(* CODESYS project Projeto_Prensa.project

Project tree, tasks and I/O mapping:
  Device : CODESYS Control Win V3, 3S - Smart Software Solutions GmbH, order no. 305021, version 3.5.11.30
    application Application
      libraries: Standard, * (System)
      task MainTask (cyclic, interval t#20ms, priority 1) calls PLC_PRG
      task VISU_TASK (cyclic, interval 100 ms, priority 31) calls VisuElems.Visu_Prg
      program PLC_PRG [LD]
      Symbols
      visualisation Visualization
  libraries: VisuSymbols, 3.5.10.0 (System)
  text list GlobalTextList
*)

// Device/Application/PLC_PRG
PROGRAM PLC_PRG
VAR
	SENSOR1: REAL; //SENSOR DE PRESSÃO M1
	SENSOR2: REAL; //SENSOR DE PRESSÃO M2
	SENSOR3: REAL; //SENSOR DE PRESSÃO P1
	PRES1: REAL; //PRESSÃO M1
	PRES2: REAL; //PRESSÃO M2
	PRES3: REAL; //PRESSÃO P1
	AL1: BOOL; // ALARME PRES1
	AL2: BOOL; // ALARME PRES2
	AL3: BOOL; // ALARME PRES3
	I7: BOOL; //B1
	I0: BOOL; //S1
	I1: BOOL; //S2
	I2: BOOL; //S3
	I3: BOOL; //S4
	I4: BOOL; //S5
	I5: BOOL; //S6
	M0: BOOL; //K1
	M1: BOOL; //K2
	M2: BOOL; //K3
	M3: BOOL; //K4
	M4: BOOL; //K5
	Q0: BOOL; //Y1
	Q1: BOOL; //Y2
	Q2: BOOL; //Y3
	Q3: BOOL; //Y4
	Q4: BOOL; //Y5
	ED0: BYTE;  // Byte para fluidsim - ENTRADAS
	AB0: BYTE;  // Byte para fluidsim - SAIDAS
END_VAR
VAR // added by the converter: edge detectors and wires of the graphical bodies
    _w1 : BOOL;
END_VAR

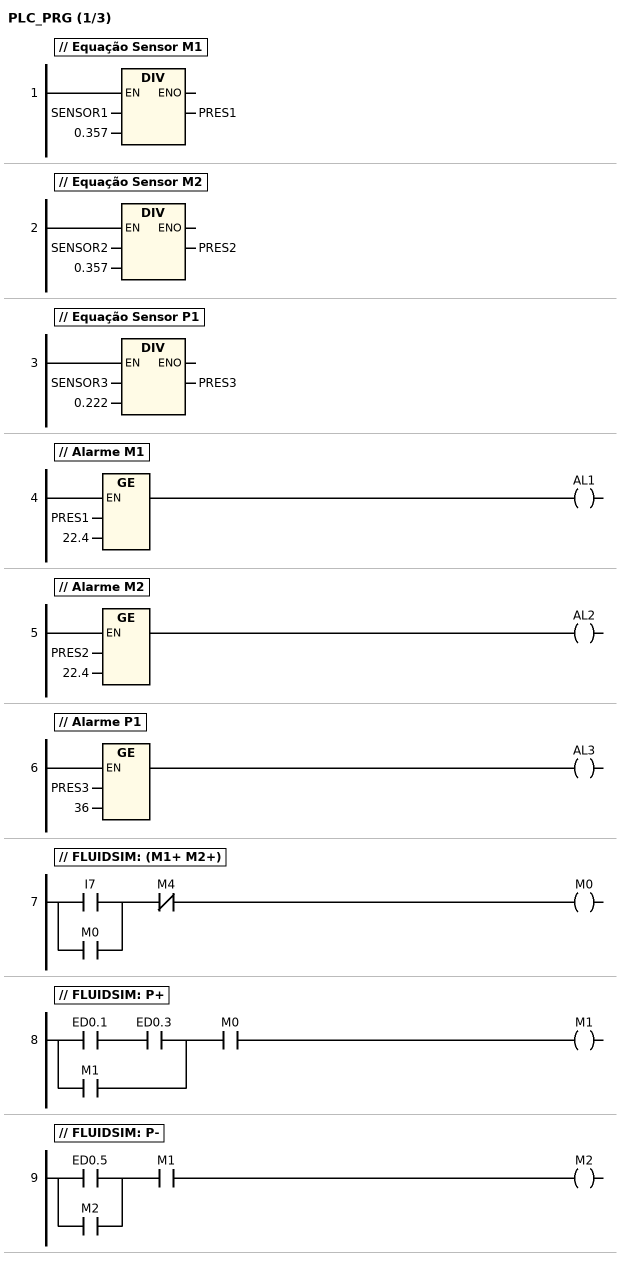
// NETWORK 1
// label: // Equação Sensor M1
PRES1 := SENSOR1 / 0.357;

// NETWORK 2
// label: // Equação Sensor M2
PRES2 := SENSOR2 / 0.357;

// NETWORK 3
// label: // Equação Sensor P1
PRES3 := SENSOR3 / 0.222;

// NETWORK 4
// label: // Alarme M1
AL1 := PRES1 >= 22.4;

// NETWORK 5
// label: // Alarme M2
AL2 := PRES2 >= 22.4;

// NETWORK 6
// label: // Alarme P1
AL3 := PRES3 >= 36;

// NETWORK 7
// label: // FLUIDSIM: (M1+ M2+)
M0 := (I7 OR M0) AND NOT M4;

// NETWORK 8
// label: // FLUIDSIM: P+
M1 := (ED0.1 AND ED0.3 OR M1) AND M0;

// NETWORK 9
// label: // FLUIDSIM: P-
M2 := (ED0.5 OR M2) AND M1;

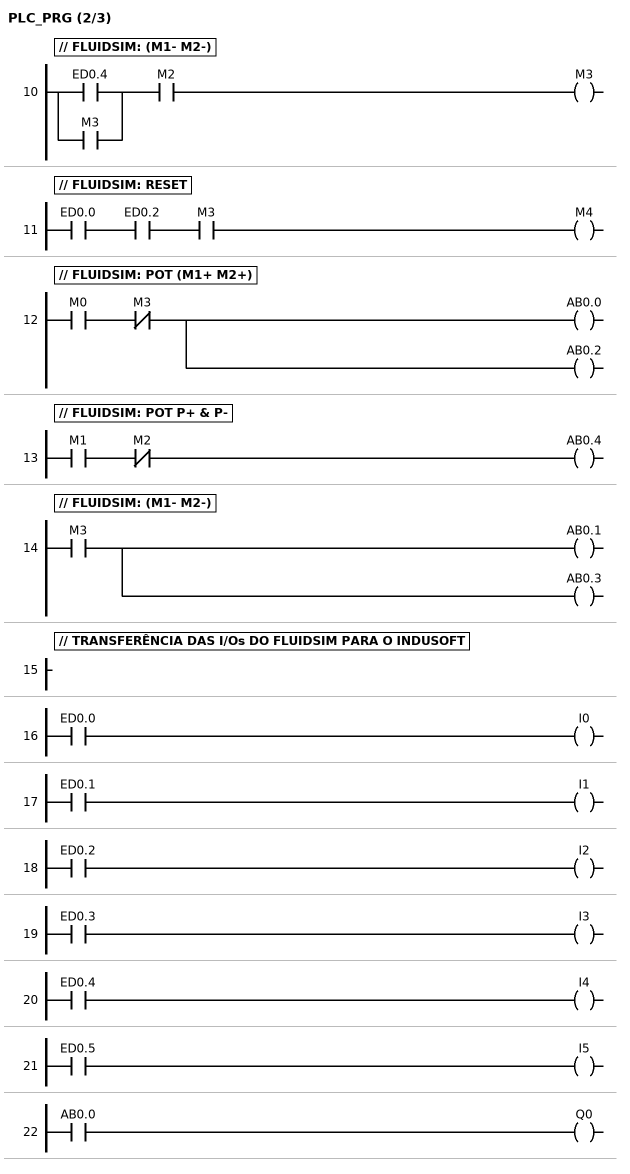
// NETWORK 10
// label: // FLUIDSIM: (M1- M2-)
M3 := (ED0.4 OR M3) AND M2;

// NETWORK 11
// label: // FLUIDSIM: RESET
M4 := ED0.0 AND ED0.2 AND M3;

// NETWORK 12
// label: // FLUIDSIM: POT (M1+ M2+)
_w1 := M0 AND NOT M3;
AB0.0 := _w1;
AB0.2 := _w1;

// NETWORK 13
// label: // FLUIDSIM: POT P+ & P-
AB0.4 := M1 AND NOT M2;

// NETWORK 14
// label: // FLUIDSIM: (M1- M2-)
AB0.1 := M3;
AB0.3 := M3;

// NETWORK 15
// label: // TRANSFERÊNCIA DAS I/Os DO FLUIDSIM PARA O INDUSOFT

// NETWORK 16
I0 := ED0.0;

// NETWORK 17
I1 := ED0.1;

// NETWORK 18
I2 := ED0.2;

// NETWORK 19
I3 := ED0.3;

// NETWORK 20
I4 := ED0.4;

// NETWORK 21
I5 := ED0.5;

// NETWORK 22
Q0 := AB0.0;

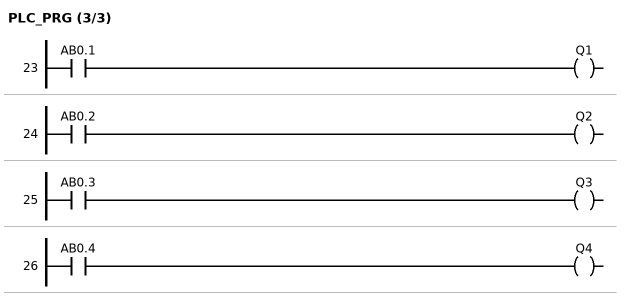
// NETWORK 23
Q1 := AB0.1;

// NETWORK 24
Q2 := AB0.2;

// NETWORK 25
Q3 := AB0.3;

// NETWORK 26
Q4 := AB0.4;

END_PROGRAM

// Device/Application/Visualization
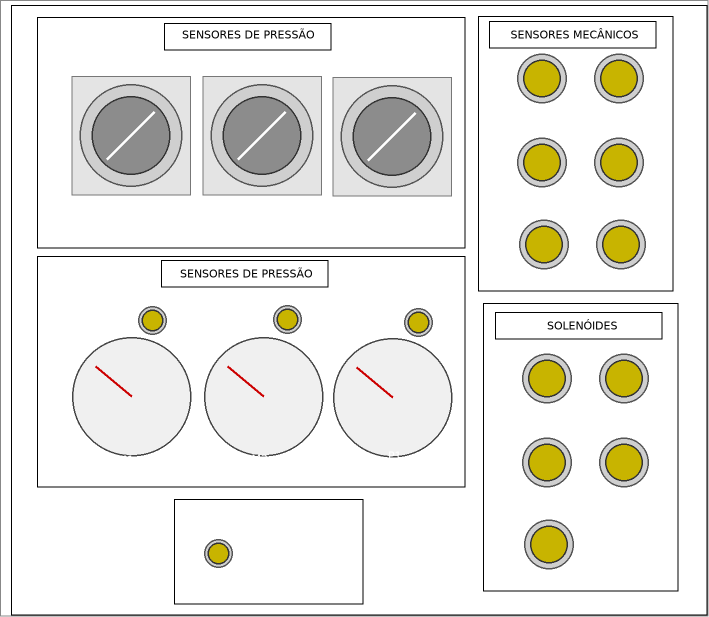
VISUALIZATION Visualization  // 709x617
    RoundedRectangle (11,5 696x610)
    RoundedRectangle (37,17 428x231)
    Potentiometer360 (57,76 148x119), variable: PLC_PRG.SENSOR1, style: Potentiometer-Potentiometer360-Gray, scale format: %.1f, scale 0..10
        p2431819421: Outside
    Potentiometer360 (188,76 148x119), variable: PLC_PRG.SENSOR2, style: Potentiometer-Potentiometer360-Gray, scale format: %.1f, scale 0..10
        p2431819421: Outside
    Potentiometer360 (318,77 148x119), variable: PLC_PRG.SENSOR3, style: Potentiometer-Potentiometer360-Gray, scale format: %.1f, scale 0..10
        p2431819421: Outside
    RoundedRectangle (478,16 195x275)
    RoundedRectangle (37,256 428x231)
    Meter90 (72,325 119x143), value: PLC_PRG.PRES1, style: Meter-Meter90-Gray, scale format: %.1f, scale 0..28
    Meter90 (204,325 119x143), value: PLC_PRG.PRES2, style: Meter-Meter90-Gray, scale format: %.1f, scale 0..28
    Meter90 (333,326 119x143), value: PLC_PRG.PRES3, style: Meter-Meter90-Gray, scale format: %.1f, scale 0..45
    Lamp1 (509,50 66x57), variable: PLC_PRG.I0, style: Lamp-Lamp1-Yellow
    Lamp1 (586,50 66x57), variable: PLC_PRG.I1, style: Lamp-Lamp1-Yellow
    Lamp1 (509,134 66x57), variable: PLC_PRG.I2, style: Lamp-Lamp1-Yellow
    Lamp1 (586,134 66x57), variable: PLC_PRG.I3, style: Lamp-Lamp1-Yellow
    Lamp1 (511,216 66x57), variable: PLC_PRG.I4, style: Lamp-Lamp1-Yellow
    Lamp1 (588,216 66x57), variable: PLC_PRG.I5, style: Lamp-Lamp1-Yellow
    RoundedRectangle (483,303 195x288)
    Lamp1 (514,350 66x57), variable: PLC_PRG.Q0, style: Lamp-Lamp1-Yellow
    Lamp1 (591,350 66x57), variable: PLC_PRG.Q1, style: Lamp-Lamp1-Yellow
    Lamp1 (514,434 66x57), variable: PLC_PRG.Q2, style: Lamp-Lamp1-Yellow
    Lamp1 (591,434 66x57), variable: PLC_PRG.Q3, style: Lamp-Lamp1-Yellow
    Lamp1 (516,516 66x57), variable: PLC_PRG.Q4, style: Lamp-Lamp1-Yellow
    RoundedRectangle (164,23 167x27)
    Label (139,20 219x30), "SENSORES DE PRESSÃO"
    RoundedRectangle (161,260 167x27)
    Label (137,259 219x30), "SENSORES DE PRESSÃO"
    RoundedRectangle (495,312 167x27)
    Label (473,311 219x30), "SOLENÓIDES"
    RoundedRectangle (489,21 167x27)
    Label (465,20 219x30), "SENSORES MECÂNICOS"
    Label (38,202 150x30), "M1"
    Label (171,203 150x30), "M2"
    Label (303,202 150x30), "P1"
    Label (462,106 150x30), "S1"
    Label (543,106 150x30), "S2"
    Label (464,187 150x30), "S3"
    Label (543,185 150x30), "S4"
    Label (465,267 150x30), "S5"
    Label (544,266 150x30), "S6"
    Label (470,402 150x30), "Y1"
    Label (545,402 150x30), "Y2"
    Label (471,485 150x30), "Y3"
    Label (547,486 150x30), "Y4"
    Label (516,530 150x30), "Y5"
    RoundedRectangle (174,499 189x105)
    Label (51,445 150x30), "M1"
    Label (185,444 150x30), "M2"
    Label (320,441 150x30), "P1"
    Lamp1 (134,304 37x33), variable: PLC_PRG.AL1, style: Lamp-Lamp1-Yellow
    Lamp1 (269,303 37x33), variable: PLC_PRG.AL2, style: Lamp-Lamp1-Yellow
    Lamp1 (400,306 37x33), variable: PLC_PRG.AL3, style: Lamp-Lamp1-Yellow
    Lamp1 (200,537 37x33), variable: PLC_PRG.I7, style: Lamp-Lamp1-Yellow
    Label (222,539 137x30), "BOTÃO - START"
END_VISUALIZATION
